FUNCTION_BLOCK fbFluentString
VAR
	_resultString : STRING(255);
END_VAR

METHOD Append : REFERENCE TO fbFluentString
VAR_INPUT
	In : STRING(255);
END_VAR
_resultString := CONCAT(_resultString, In);
Append REF= THIS^;
END_METHOD

PROPERTY Result : STRING(255)
GET
Result := _resultString;
_resultString := '';
END_GET
SET
END_SET
END_PROPERTY

END_FUNCTION_BLOCK

(* stored: Version 1.1.0.1, ProductVersion 3.1.4024.2
   POU fbFluentString: Id {8476f40e-c0b0-41f8-be7d-ef76ddbbb55b}, SpecialFunc None
   Method Append: Id {9d22aabf-8fd1-44ed-abaa-ad13dea6b117}
   Property Result: Id {dc40d10e-1859-4a54-8a27-9aeb12aba65d}
   Get Get: Id {cc4065a5-546d-47eb-8dd1-610c0cb72af3}
   Set Set: Id {16a8541c-69aa-41e4-8241-9b177b343926} *)
